# EPICS autosave request: ADApp/Db/NDTimeSeries_settings.req
$(P)$(R)TSNumPoints
$(P)$(R)TSRead.SCAN
$(P)$(R)TSAcquireMode
$(P)$(R)TSComputeFFT
file "NDPluginBase_settings.req", P=$(P), R=$(R)
